TYPE ST_Energy :
STRUCT
END_STRUCT
END_TYPE

(* stored: Version 1.1.0.1, ProductVersion 3.1.4024.5
   DUT ST_Energy: Id {b68dd15d-02c8-4fa5-b6af-0039fa3db41d} *)
